INTERFACE I_FBDiag

PROPERTY P_diagBits : st_diagFBBits
GET
END_GET
END_PROPERTY

PROPERTY P_State : STRING(20)
GET
END_GET
END_PROPERTY

END_INTERFACE

(* stored: Version 1.1.0.1, ProductVersion 3.1.4024.12
   Itf I_FBDiag: Id {04f94619-e2a7-46c6-ac37-08520c68d83a}
   Property P_diagBits: Id {becec5d2-04e3-4f2a-a307-040fc135c7b9}
   Get Get: Id {d92f5385-dabc-4135-a091-f06766c729a3}
   Property P_State: Id {fbb64f56-6859-4630-978d-ec6ce0932419}
   Get Get: Id {4ff4aeb3-fd3f-4d7a-821d-c92ea22ee184} *)
